// TIA Portal V20 export
FUNCTION "CallManualOperationLines_CITI" : Void   // FC183, LAD
// stored: Access Published, SetENOAutomatically false
   VAR_TEMP
      status : Array[0..30] of Word;   // Status of the Blocks
      errorID : Array[0..30] of Word;   // Error IDs of the Blocks
      call_index : Int;
   END_VAR
   VAR CONSTANT
      MECHANIC_NAME_ENABLE : Bool := FALSE;   // Activation of the Mechanic names
   END_VAR
BEGIN

REGION Network 1: CITI Manual Lines Configuration
   // Equipment Module 3400
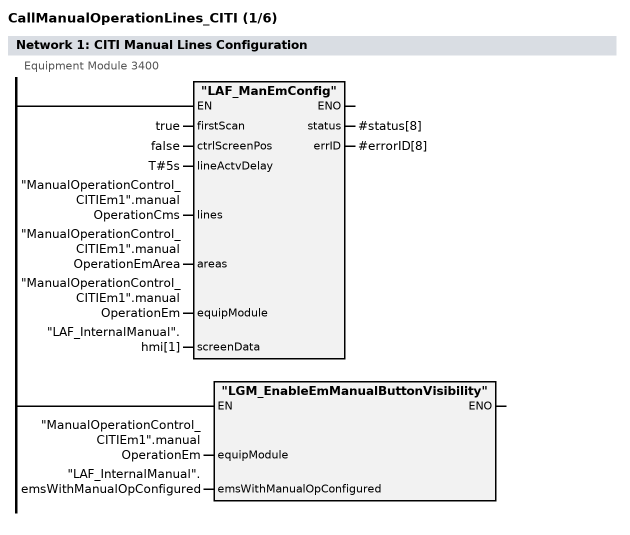
   RUNG wire#powerrail
      "LAF_ManEmConfig"(firstScan := true, ctrlScreenPos := false, lineActvDelay := T#5s, lines := "ManualOperationControl_CITIEm1".manualOperationCms, areas := "ManualOperationControl_CITIEm1".manualOperationEmArea, equipModule := "ManualOperationControl_CITIEm1".manualOperationEm, screenData := "LAF_InternalManual".hmi[1], status => #status[8], errID => #errorID[8])
   END_RUNG
   RUNG wire#powerrail
      "LGM_EnableEmManualButtonVisibility"(equipModule := "ManualOperationControl_CITIEm1".manualOperationEm, emsWithManualOpConfigured := "LAF_InternalManual".emsWithManualOpConfigured)
   END_RUNG
   // the same network as SCL:
   "LAF_ManEmConfig"(firstScan := true,
                     ctrlScreenPos := false,
                     lineActvDelay := T#5s,
                     lines := "ManualOperationControl_CITIEm1".manualOperationCms,
                     areas := "ManualOperationControl_CITIEm1".manualOperationEmArea,
                     equipModule := "ManualOperationControl_CITIEm1".manualOperationEm,
                     screenData := "LAF_InternalManual".hmi[1],
                     status => #status[8],
                     errID => #errorID[8]);
   "LGM_EnableEmManualButtonVisibility"(equipModule := "ManualOperationControl_CITIEm1".manualOperationEm,
                           emsWithManualOpConfigured := "LAF_InternalManual".emsWithManualOpConfigured);
END_REGION

REGION Network 2: CITI1 Equipment Module 1 Line 1
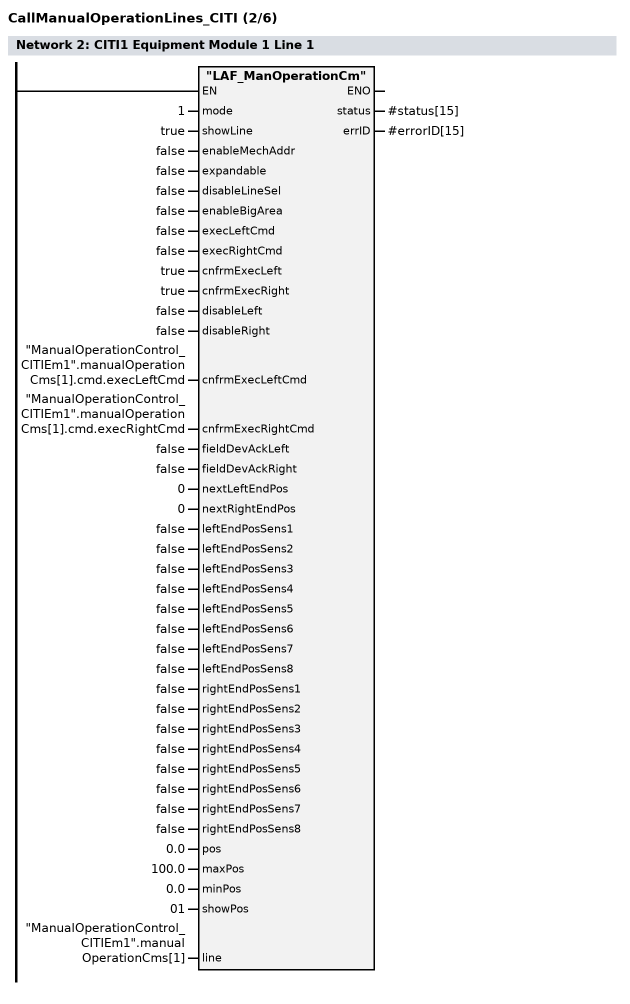
   RUNG wire#powerrail
      "LAF_ManOperationCm"(mode := 1, showLine := true, enableMechAddr := false, expandable := false, disableLineSel := false, enableBigArea := false, execLeftCmd := false, execRightCmd := false, cnfrmExecLeft := true, cnfrmExecRight := true, disableLeft := false, disableRight := false, cnfrmExecLeftCmd := "ManualOperationControl_CITIEm1".manualOperationCms[1].cmd.execLeftCmd, cnfrmExecRightCmd := "ManualOperationControl_CITIEm1".manualOperationCms[1].cmd.execRightCmd, fieldDevAckLeft := false, fieldDevAckRight := false, nextLeftEndPos := 0, nextRightEndPos := 0, leftEndPosSens1 := false, leftEndPosSens2 := false, leftEndPosSens3 := false, leftEndPosSens4 := false, leftEndPosSens5 := false, leftEndPosSens6 := false, leftEndPosSens7 := false, leftEndPosSens8 := false, rightEndPosSens1 := false, rightEndPosSens2 := false, rightEndPosSens3 := false, rightEndPosSens4 := false, rightEndPosSens5 := false, rightEndPosSens6 := false, rightEndPosSens7 := false, rightEndPosSens8 := false, pos := 0.0, maxPos := 100.0, minPos := 0.0, showPos := 01, line := "ManualOperationControl_CITIEm1".manualOperationCms[1], status => #status[15], errID => #errorID[15])
   END_RUNG
   // the same network as SCL:
   "LAF_ManOperationCm"(mode := 1,
                        showLine := true,
                        enableMechAddr := false,
                        expandable := false,
                        disableLineSel := false,
                        enableBigArea := false,
                        execLeftCmd := false,
                        execRightCmd := false,
                        cnfrmExecLeft := true,
                        cnfrmExecRight := true,
                        disableLeft := false,
                        disableRight := false,
                        cnfrmExecLeftCmd := "ManualOperationControl_CITIEm1".manualOperationCms[1].cmd.execLeftCmd,
                        cnfrmExecRightCmd := "ManualOperationControl_CITIEm1".manualOperationCms[1].cmd.execRightCmd,
                        fieldDevAckLeft := false,
                        fieldDevAckRight := false,
                        nextLeftEndPos := 0,
                        nextRightEndPos := 0,
                        leftEndPosSens1 := false,
                        leftEndPosSens2 := false,
                        leftEndPosSens3 := false,
                        leftEndPosSens4 := false,
                        leftEndPosSens5 := false,
                        leftEndPosSens6 := false,
                        leftEndPosSens7 := false,
                        leftEndPosSens8 := false,
                        rightEndPosSens1 := false,
                        rightEndPosSens2 := false,
                        rightEndPosSens3 := false,
                        rightEndPosSens4 := false,
                        rightEndPosSens5 := false,
                        rightEndPosSens6 := false,
                        rightEndPosSens7 := false,
                        rightEndPosSens8 := false,
                        pos := 0.0,
                        maxPos := 100.0,
                        minPos := 0.0,
                        showPos := 01,
                        line := "ManualOperationControl_CITIEm1".manualOperationCms[1],
                        status => #status[15],
                        errID => #errorID[15]);
END_REGION

REGION Network 3: CITI1 Equipment Module 1 Line 2
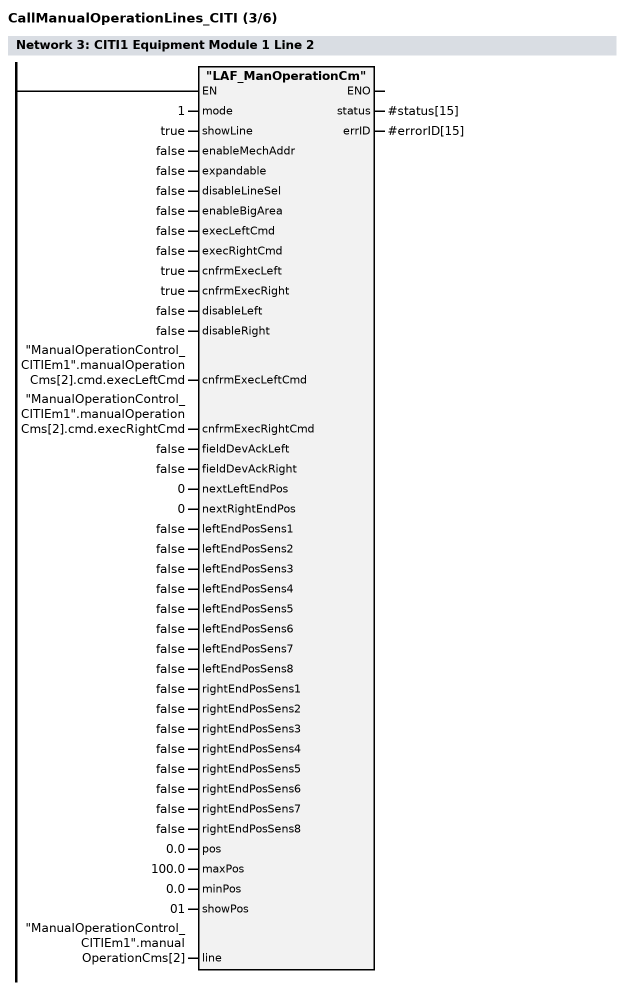
   RUNG wire#powerrail
      "LAF_ManOperationCm"(mode := 1, showLine := true, enableMechAddr := false, expandable := false, disableLineSel := false, enableBigArea := false, execLeftCmd := false, execRightCmd := false, cnfrmExecLeft := true, cnfrmExecRight := true, disableLeft := false, disableRight := false, cnfrmExecLeftCmd := "ManualOperationControl_CITIEm1".manualOperationCms[2].cmd.execLeftCmd, cnfrmExecRightCmd := "ManualOperationControl_CITIEm1".manualOperationCms[2].cmd.execRightCmd, fieldDevAckLeft := false, fieldDevAckRight := false, nextLeftEndPos := 0, nextRightEndPos := 0, leftEndPosSens1 := false, leftEndPosSens2 := false, leftEndPosSens3 := false, leftEndPosSens4 := false, leftEndPosSens5 := false, leftEndPosSens6 := false, leftEndPosSens7 := false, leftEndPosSens8 := false, rightEndPosSens1 := false, rightEndPosSens2 := false, rightEndPosSens3 := false, rightEndPosSens4 := false, rightEndPosSens5 := false, rightEndPosSens6 := false, rightEndPosSens7 := false, rightEndPosSens8 := false, pos := 0.0, maxPos := 100.0, minPos := 0.0, showPos := 01, line := "ManualOperationControl_CITIEm1".manualOperationCms[2], status => #status[15], errID => #errorID[15])
   END_RUNG
   // the same network as SCL:
   "LAF_ManOperationCm"(mode := 1,
                        showLine := true,
                        enableMechAddr := false,
                        expandable := false,
                        disableLineSel := false,
                        enableBigArea := false,
                        execLeftCmd := false,
                        execRightCmd := false,
                        cnfrmExecLeft := true,
                        cnfrmExecRight := true,
                        disableLeft := false,
                        disableRight := false,
                        cnfrmExecLeftCmd := "ManualOperationControl_CITIEm1".manualOperationCms[2].cmd.execLeftCmd,
                        cnfrmExecRightCmd := "ManualOperationControl_CITIEm1".manualOperationCms[2].cmd.execRightCmd,
                        fieldDevAckLeft := false,
                        fieldDevAckRight := false,
                        nextLeftEndPos := 0,
                        nextRightEndPos := 0,
                        leftEndPosSens1 := false,
                        leftEndPosSens2 := false,
                        leftEndPosSens3 := false,
                        leftEndPosSens4 := false,
                        leftEndPosSens5 := false,
                        leftEndPosSens6 := false,
                        leftEndPosSens7 := false,
                        leftEndPosSens8 := false,
                        rightEndPosSens1 := false,
                        rightEndPosSens2 := false,
                        rightEndPosSens3 := false,
                        rightEndPosSens4 := false,
                        rightEndPosSens5 := false,
                        rightEndPosSens6 := false,
                        rightEndPosSens7 := false,
                        rightEndPosSens8 := false,
                        pos := 0.0,
                        maxPos := 100.0,
                        minPos := 0.0,
                        showPos := 01,
                        line := "ManualOperationControl_CITIEm1".manualOperationCms[2],
                        status => #status[15],
                        errID => #errorID[15]);
END_REGION

REGION Network 4: CITI1 Equipment Module 1 Line 3
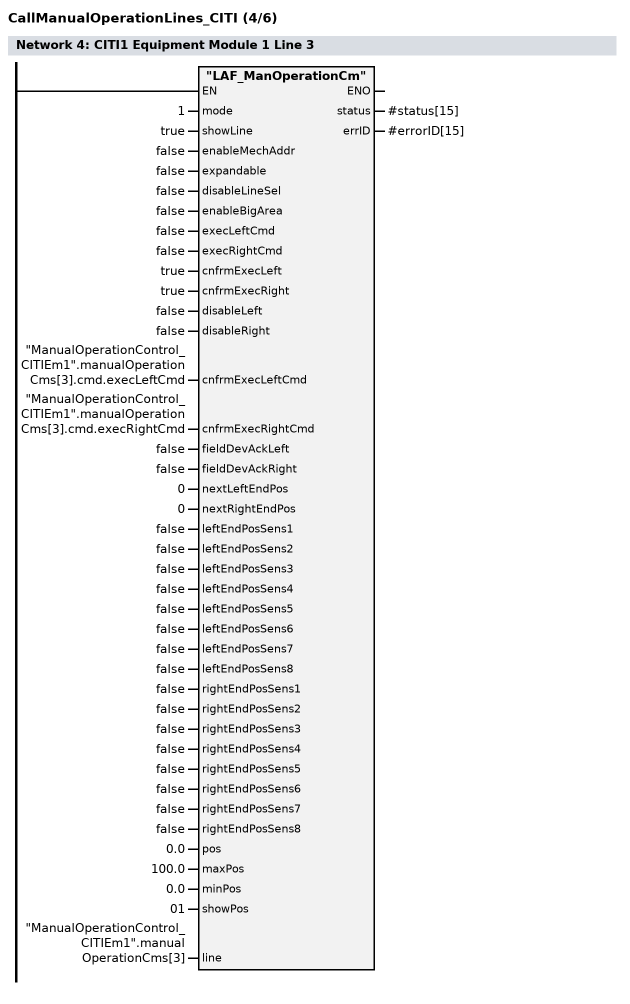
   RUNG wire#powerrail
      "LAF_ManOperationCm"(mode := 1, showLine := true, enableMechAddr := false, expandable := false, disableLineSel := false, enableBigArea := false, execLeftCmd := false, execRightCmd := false, cnfrmExecLeft := true, cnfrmExecRight := true, disableLeft := false, disableRight := false, cnfrmExecLeftCmd := "ManualOperationControl_CITIEm1".manualOperationCms[3].cmd.execLeftCmd, cnfrmExecRightCmd := "ManualOperationControl_CITIEm1".manualOperationCms[3].cmd.execRightCmd, fieldDevAckLeft := false, fieldDevAckRight := false, nextLeftEndPos := 0, nextRightEndPos := 0, leftEndPosSens1 := false, leftEndPosSens2 := false, leftEndPosSens3 := false, leftEndPosSens4 := false, leftEndPosSens5 := false, leftEndPosSens6 := false, leftEndPosSens7 := false, leftEndPosSens8 := false, rightEndPosSens1 := false, rightEndPosSens2 := false, rightEndPosSens3 := false, rightEndPosSens4 := false, rightEndPosSens5 := false, rightEndPosSens6 := false, rightEndPosSens7 := false, rightEndPosSens8 := false, pos := 0.0, maxPos := 100.0, minPos := 0.0, showPos := 01, line := "ManualOperationControl_CITIEm1".manualOperationCms[3], status => #status[15], errID => #errorID[15])
   END_RUNG
   // the same network as SCL:
   "LAF_ManOperationCm"(mode := 1,
                        showLine := true,
                        enableMechAddr := false,
                        expandable := false,
                        disableLineSel := false,
                        enableBigArea := false,
                        execLeftCmd := false,
                        execRightCmd := false,
                        cnfrmExecLeft := true,
                        cnfrmExecRight := true,
                        disableLeft := false,
                        disableRight := false,
                        cnfrmExecLeftCmd := "ManualOperationControl_CITIEm1".manualOperationCms[3].cmd.execLeftCmd,
                        cnfrmExecRightCmd := "ManualOperationControl_CITIEm1".manualOperationCms[3].cmd.execRightCmd,
                        fieldDevAckLeft := false,
                        fieldDevAckRight := false,
                        nextLeftEndPos := 0,
                        nextRightEndPos := 0,
                        leftEndPosSens1 := false,
                        leftEndPosSens2 := false,
                        leftEndPosSens3 := false,
                        leftEndPosSens4 := false,
                        leftEndPosSens5 := false,
                        leftEndPosSens6 := false,
                        leftEndPosSens7 := false,
                        leftEndPosSens8 := false,
                        rightEndPosSens1 := false,
                        rightEndPosSens2 := false,
                        rightEndPosSens3 := false,
                        rightEndPosSens4 := false,
                        rightEndPosSens5 := false,
                        rightEndPosSens6 := false,
                        rightEndPosSens7 := false,
                        rightEndPosSens8 := false,
                        pos := 0.0,
                        maxPos := 100.0,
                        minPos := 0.0,
                        showPos := 01,
                        line := "ManualOperationControl_CITIEm1".manualOperationCms[3],
                        status => #status[15],
                        errID => #errorID[15]);
END_REGION

REGION Network 5: CITI1 Equipment Module 1 Line 4
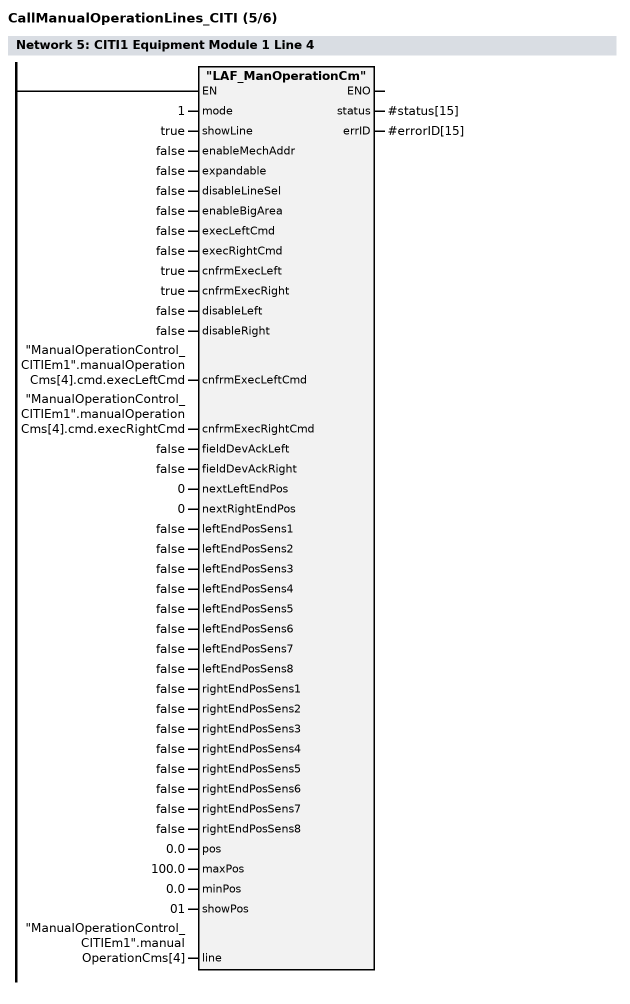
   RUNG wire#powerrail
      "LAF_ManOperationCm"(mode := 1, showLine := true, enableMechAddr := false, expandable := false, disableLineSel := false, enableBigArea := false, execLeftCmd := false, execRightCmd := false, cnfrmExecLeft := true, cnfrmExecRight := true, disableLeft := false, disableRight := false, cnfrmExecLeftCmd := "ManualOperationControl_CITIEm1".manualOperationCms[4].cmd.execLeftCmd, cnfrmExecRightCmd := "ManualOperationControl_CITIEm1".manualOperationCms[4].cmd.execRightCmd, fieldDevAckLeft := false, fieldDevAckRight := false, nextLeftEndPos := 0, nextRightEndPos := 0, leftEndPosSens1 := false, leftEndPosSens2 := false, leftEndPosSens3 := false, leftEndPosSens4 := false, leftEndPosSens5 := false, leftEndPosSens6 := false, leftEndPosSens7 := false, leftEndPosSens8 := false, rightEndPosSens1 := false, rightEndPosSens2 := false, rightEndPosSens3 := false, rightEndPosSens4 := false, rightEndPosSens5 := false, rightEndPosSens6 := false, rightEndPosSens7 := false, rightEndPosSens8 := false, pos := 0.0, maxPos := 100.0, minPos := 0.0, showPos := 01, line := "ManualOperationControl_CITIEm1".manualOperationCms[4], status => #status[15], errID => #errorID[15])
   END_RUNG
   // the same network as SCL:
   "LAF_ManOperationCm"(mode := 1,
                        showLine := true,
                        enableMechAddr := false,
                        expandable := false,
                        disableLineSel := false,
                        enableBigArea := false,
                        execLeftCmd := false,
                        execRightCmd := false,
                        cnfrmExecLeft := true,
                        cnfrmExecRight := true,
                        disableLeft := false,
                        disableRight := false,
                        cnfrmExecLeftCmd := "ManualOperationControl_CITIEm1".manualOperationCms[4].cmd.execLeftCmd,
                        cnfrmExecRightCmd := "ManualOperationControl_CITIEm1".manualOperationCms[4].cmd.execRightCmd,
                        fieldDevAckLeft := false,
                        fieldDevAckRight := false,
                        nextLeftEndPos := 0,
                        nextRightEndPos := 0,
                        leftEndPosSens1 := false,
                        leftEndPosSens2 := false,
                        leftEndPosSens3 := false,
                        leftEndPosSens4 := false,
                        leftEndPosSens5 := false,
                        leftEndPosSens6 := false,
                        leftEndPosSens7 := false,
                        leftEndPosSens8 := false,
                        rightEndPosSens1 := false,
                        rightEndPosSens2 := false,
                        rightEndPosSens3 := false,
                        rightEndPosSens4 := false,
                        rightEndPosSens5 := false,
                        rightEndPosSens6 := false,
                        rightEndPosSens7 := false,
                        rightEndPosSens8 := false,
                        pos := 0.0,
                        maxPos := 100.0,
                        minPos := 0.0,
                        showPos := 01,
                        line := "ManualOperationControl_CITIEm1".manualOperationCms[4],
                        status => #status[15],
                        errID => #errorID[15]);
END_REGION

REGION Network 6: CITI1 Equipment Module 1 Line 5
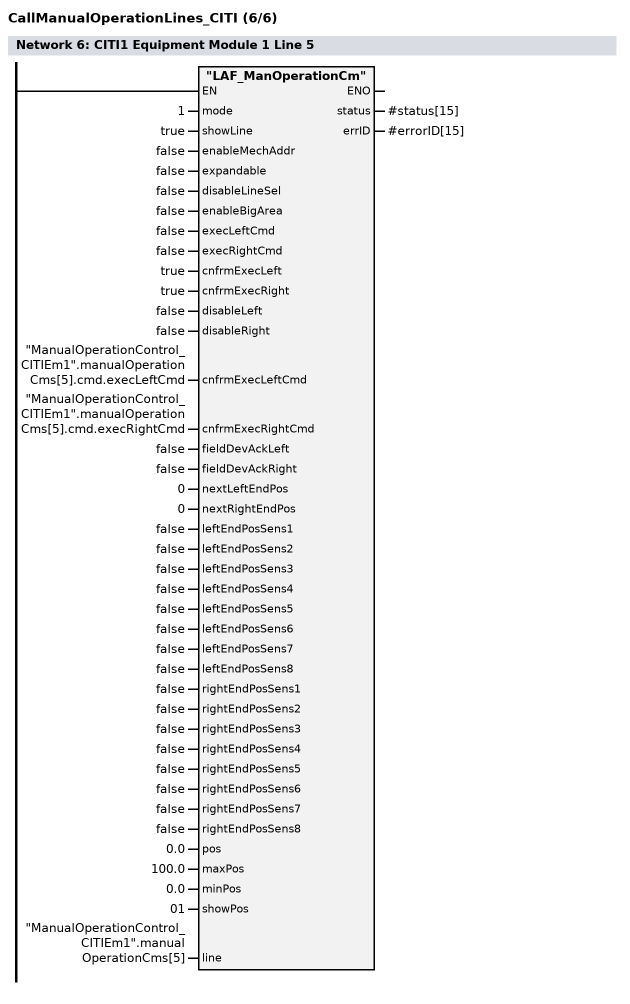
   RUNG wire#powerrail
      "LAF_ManOperationCm"(mode := 1, showLine := true, enableMechAddr := false, expandable := false, disableLineSel := false, enableBigArea := false, execLeftCmd := false, execRightCmd := false, cnfrmExecLeft := true, cnfrmExecRight := true, disableLeft := false, disableRight := false, cnfrmExecLeftCmd := "ManualOperationControl_CITIEm1".manualOperationCms[5].cmd.execLeftCmd, cnfrmExecRightCmd := "ManualOperationControl_CITIEm1".manualOperationCms[5].cmd.execRightCmd, fieldDevAckLeft := false, fieldDevAckRight := false, nextLeftEndPos := 0, nextRightEndPos := 0, leftEndPosSens1 := false, leftEndPosSens2 := false, leftEndPosSens3 := false, leftEndPosSens4 := false, leftEndPosSens5 := false, leftEndPosSens6 := false, leftEndPosSens7 := false, leftEndPosSens8 := false, rightEndPosSens1 := false, rightEndPosSens2 := false, rightEndPosSens3 := false, rightEndPosSens4 := false, rightEndPosSens5 := false, rightEndPosSens6 := false, rightEndPosSens7 := false, rightEndPosSens8 := false, pos := 0.0, maxPos := 100.0, minPos := 0.0, showPos := 01, line := "ManualOperationControl_CITIEm1".manualOperationCms[5], status => #status[15], errID => #errorID[15])
   END_RUNG
   // the same network as SCL:
   "LAF_ManOperationCm"(mode := 1,
                        showLine := true,
                        enableMechAddr := false,
                        expandable := false,
                        disableLineSel := false,
                        enableBigArea := false,
                        execLeftCmd := false,
                        execRightCmd := false,
                        cnfrmExecLeft := true,
                        cnfrmExecRight := true,
                        disableLeft := false,
                        disableRight := false,
                        cnfrmExecLeftCmd := "ManualOperationControl_CITIEm1".manualOperationCms[5].cmd.execLeftCmd,
                        cnfrmExecRightCmd := "ManualOperationControl_CITIEm1".manualOperationCms[5].cmd.execRightCmd,
                        fieldDevAckLeft := false,
                        fieldDevAckRight := false,
                        nextLeftEndPos := 0,
                        nextRightEndPos := 0,
                        leftEndPosSens1 := false,
                        leftEndPosSens2 := false,
                        leftEndPosSens3 := false,
                        leftEndPosSens4 := false,
                        leftEndPosSens5 := false,
                        leftEndPosSens6 := false,
                        leftEndPosSens7 := false,
                        leftEndPosSens8 := false,
                        rightEndPosSens1 := false,
                        rightEndPosSens2 := false,
                        rightEndPosSens3 := false,
                        rightEndPosSens4 := false,
                        rightEndPosSens5 := false,
                        rightEndPosSens6 := false,
                        rightEndPosSens7 := false,
                        rightEndPosSens8 := false,
                        pos := 0.0,
                        maxPos := 100.0,
                        minPos := 0.0,
                        showPos := 01,
                        line := "ManualOperationControl_CITIEm1".manualOperationCms[5],
                        status => #status[15],
                        errID => #errorID[15]);
END_REGION
END_FUNCTION
